// TwinCAT 3 PLC project Untitled1
// ProgramVersion: 3.1.4024.0
// libraries:
//   Tc2_Math, * (Beckhoff Automation GmbH)
//   Tc2_Standard, * (Beckhoff Automation GmbH)
//   Tc2_System, * (Beckhoff Automation GmbH)
//   Tc3_Mc3PlanarMotion, * (Beckhoff Automation GmbH)
//   Tc3_Module, * (Beckhoff Automation GmbH)
//   Tc3_Physics, * (Beckhoff Automation GmbH)
//   XboxControllerUtilities, * (Beckhoff Community)
// project tree:
//   Configuration/ Constraints.TcGVL
//   Mover/ Planar_Mover.TcPOU
//   / PlcTask.TcTTO
//   Controller/ XboxController.TcPOU
// real-time tasks:
//   TASK PlcTask: cycle T#10ms, priority 20, ADS port 350

CONFIGURATION Untitled1
    RESOURCE PLC ON TwinCAT3
        TASK PlcTask(INTERVAL := T#10ms, PRIORITY := 20);
        PROGRAM XboxController WITH PlcTask : XboxController;
        PROGRAM Planar_Mover WITH PlcTask : Planar_Mover;
    END_RESOURCE
END_CONFIGURATION

// ---- Configuration/Constraints.TcGVL
{attribute 'qualified_only'}
VAR_GLOBAL
	

	deltaT						: 		LREAL 	:= 0.000250 ; 	// Cycle time of PLC in Seconds
	maxVelocity					: 		LREAL	:= 150;			// mm/s
	Kp 							:		LREAL      := 3; 		// P Term
	Ki 							:		LREAL      := 0.5; 		// I Term
	Kd 							:		LREAL      := 2; 		// D Term
	Restarting					: 		BOOL;
	
	
END_VAR

// ---- Controller/XboxController.TcPOU
PROGRAM XboxController
VAR

	XboxController1 			: 		FB_Xbox_Controller(NetID := '', iControllerNumber := 1);	
	bIsConnected   				:  		ARRAY [1..2] OF BOOL;
	XpPosition					:		ARRAY [1..2] OF MoverVector; 
	MoverPos					: 		ARRAY [1..2] OF MoverVector;
	invertX						: 		LREAL;
	invertY						: 		LREAL;
	DestinationX				: 		DINT;
	DestinationY				: 		DINT;
	NearestRotationPoint		: 		PositionXYC;
	RotationScailing			: 		LREAL := 0.0002;
	StartTimer					: 		BOOL;
	Timer						: 		TON;
	SnapVAR						: 		BOOL;
	C_VALUE						: 		LREAL;
	MODDED_C					: 		LREAL;
	MoveToC						: 		LREAL;
	ShortestCMove				: 		PositionXYC;
	START						: 		BOOL;
	Ready						: 		BOOL; 
	
	
	
	SanitizedX					: 		LREAL;
	SanitizedY					: 		LREAL;
	SetPointX					: 		REAL;
	SetPointY					: 		REAL;
	ControllerP_Err_X			: 		LREAL;
	ControllerI_Err_X			: 		LREAL;
	ControllerD_Err_X			: 		LREAL;
	ControllerP_Err_Y			: 		LREAL;
	ControllerI_Err_Y			: 		LREAL;
	ControllerD_Err_Y			: 		LREAL;
	PrevSetPointX	 			: 		LREAL;
	PrevSetPointY	 			: 		LREAL;
	PrevSanitizedX				: 		LREAL;
	PrevSanitizedY				: 		LREAL;
	MaxRateOfChange				: 		LREAL;
	IntegralLimit				: 		LREAL;
	MaxIntegralError			: 		LREAL;
	OutputMagnitude				: 		LREAL;
	OutputDirection				: 		LREAL;
	PrevOutputMagnitude			: 		LREAL;
	OutputDistance				: 		LREAL;
	ZeroVector 					: 		MoverVector ;
	nCase						: 		INT := 1;
	Alpha						: 		LREAL := 0.01;
	MaxVelocity					:		LREAL := 10; 
	PastPos10					: 		BOOL;
	PastNeg10					: 		BOOL; 
	BOOL1                       :       BOOL;	
	BOOL2                       :       BOOL;	
	BOOL3						:       BOOL;
	XPoint						: 		BOOL;
	YPoint						: 		BOOL;	
	Height 						: 		LREAL := 2; 
	RESET						:	 	BOOL;
	Go							:		BOOL;
	R_TRIG1						: 		R_TRIG;
	R_TRIG2						: 		R_TRIG;
	SmoothingTon1				:		TON;
	SmoothingTon2				:		TON;
	Ton1						:		TON;
	Ton2						:		TON;
	TRIGGER1					: 		BOOL;
	TRIGGER2					: 		BOOL;
	XPos						: 		INT;
	YPos						: 		INT;
	MaxPosRot					: 		LREAL;
	MaxNegRot					: 		LREAL;
	filtered_output				:	 	LREAL;
	ramp_factor: LREAL;
	ramped_input: LREAL;
	GraphVar: LREAL;
		Prevoutput: LREAL;
		PrevNegRot: LREAL;
	PrevPosRot: LREAL;
		CheckNegRot: LREAL;
	CheckPosRot: LREAL;
		IsUpdated: BOOL;
			Closest90: LREAL;
	
	

END_VAR

//Xbox Controller 1 
XboxController1.Cycle();
bIsConnected[1] := XboxController1.P_Status.bConnected; 

MoverPos[1] := Planar_Mover.fbMover[1].MCTOPLC.ACT.ActPos;

IF Planar_Mover.Done AND NOT ready THEN
	XboxController.init();
END_IF

SetPoint();
		Planar_Mover.fbMover[1].SetExternalSetpoint( XPPosition[1], ZeroVector, ZeroVector);
		
Tilt();
Rotation(); 
ButtonXY();
ButtonA(); 
Bumpers();

METHOD Bumpers 
VAR_INPUT
END_VAR
VAR 
END_VAR

//Hold down for automatic raise and lowering

TON1(IN := XboxController1.P_Buttons.bLeft_Shoulder, PT := T#0.5S); 
TON2(IN := XboxController1.P_Buttons.bRight_Shoulder, PT := T#0.5S); 

IF TON1.Q THEN
	SmoothingTon1.IN := TRUE AND NOT SmoothingTon1.Q;
ELSE
	SmoothingTon1.IN := FALSE;		
END_IF

IF TON2.Q THEN
	SmoothingTon2.IN := TRUE AND NOT SmoothingTon2.Q;
ELSE
	SmoothingTon2.IN := FALSE;
END_IF

//OSR to make sure only one is seen per click 
R_TRIG1(CLK:=XboxController1.P_Buttons.bLeft_Shoulder , Q=> );
R_TRIG2(CLK:=XboxController1.P_Buttons.bRight_Shoulder, Q=> );

IF (R_TRIG1.Q OR SmoothingTon1.Q) AND Height >= -0.35 THEN 
	Height :=  Height - 0.15;
ELSIF (R_TRIG2.Q OR SmoothingTon2.Q) AND Height < 5.0 THEN
	Height := Height + 0.15;
ELSE
	Height := Height; 
END_IF

XpPosition[1].z := Height; 


SmoothingTon1.PT:=T#0.1S;
SmoothingTon2.PT:=T#0.1S;

SmoothingTON1();
SmoothingTON2();
END_METHOD

METHOD buttonA : LREAL
VAR_INPUT
END_VAR
IF XboxController.Ready AND NOT PLanar_Mover.fbMover[1].Error THEN
		
		//Rotation Handeling
		// Find Nearest X
		IF LREAL_TO_INT(MoverPos[1].X) MOD 120 < 60 THEN
			DestinationX	:= 120 * MODTURNS( MoverPos[1].X , 120 );
		ELSE
			DestinationX	:= 120 * (MODTURNS( MoverPos[1].X, 120 ) + 1);
		END_IF
		
		// Find Nearest Y
		IF LREAL_TO_INT(MoverPos[1].Y) MOD 120 < 60 THEN
			DestinationY	:= 120 * MODTURNS( MoverPos[1].Y , 120 );
		ELSE
			DestinationY	:= 120 * (MODTURNS( MoverPos[1].Y, 120 ) + 1);
		END_IF
		
		//Set Boundries for X
		IF DestinationX = 0 THEN
			DestinationX := DestinationX + 120;
		ELSIF DestinationX = 960 THEN
			DestinationX := DestinationX - 120;
		END_IF 	
		
		//Set Boundries for Y
		IF DestinationY = 0 THEN 
			DestinationY := DestinationY + 120;
		ELSIF DestinationY = 720 THEN
			DestinationY := DestinationY - 120;
		END_IF 

		//Move to Nearest Rotation point
			IF XBoxController1.P_Buttons.bA_Button AND MoverPos[1].X < DestinationX THEN
				XpPosition[1].X := XpPosition[1].X + ( 40 * Constraints.deltaT );
			ELSIF XBoxController1.P_Buttons.bA_Button AND MoverPos[1].X > DestinationX THEN
				XpPosition[1].X := XpPosition[1].X -( 40 * Constraints.deltaT );
			END_IF;
			
			IF XBoxController1.P_Buttons.bA_Button AND MoverPos[1].Y < DestinationY THEN
				XpPosition[1].Y := XpPosition[1].Y + ( 40 * Constraints.deltaT );
			ELSIF XBoxController1.P_Buttons.bA_Button AND MoverPos[1].Y > DestinationY THEN
				XpPosition[1].Y := XpPosition[1].Y -( 40 * Constraints.deltaT );
			END_IF;
	
			
			//Checking to make sure Tile is within 1 mm +- of a point that is modulo by 120 and = 0 and then truning a bool true or false
			IF ((LREAL_TO_INT(MoverPos[1].x) MOD 120) >= 119) OR ((LREAL_TO_INT(MoverPos[1].x) MOD 120) <= 1)  THEN
				XPOint := TRUE; 
			ELSE 
				XPoint := FALSE; 
			END_IF
			
			IF ((LREAL_TO_INT(MoverPos[1].y) MOD 120) >= 119) OR ((LREAL_TO_INT(MoverPos[1].y) MOD 120) <= 1) THEN
				YPOint := TRUE; 
			ELSE
				YPoint := FALSE;
			END_IF	
		
		
END_IF
END_METHOD

METHOD buttonXY : LREAL
VAR_INPUT
END_VAR
IF XboxController.Ready AND NOT PLanar_Mover.fbMover[1].Error THEN
	

			//Lock into X movement
		IF XboxController1.P_Buttons.bX_Button THEN
			XpPosition[1].y := XpPosition[1].y ;
		ELSE
			//
		END_IF
		
		//Lock into Y movement
		IF XboxController1.P_Buttons.bY_Button THEN
			XpPosition[1].x := XpPosition[1].x ;
		ELSE
			//
		END_IF
END_IF
END_METHOD

METHOD init 
VAR_INPUT
END_VAR

VAR




END_VAR

IF Planar_mover.MoverState = 3 THEN
	CASE nCase OF 
	1:
		IF Constraints.Restarting THEN
			Constraints.Restarting := FALSE;
			nCase := 4;
		//Wait to Start 
		ELSIF XboxController1.P_Buttons.bStart OR START THEN
			Start := FALSE;
			nCase := 2;
		END_IF
	
	2:
	
	
		//Mover to Play positions
		Planar_Mover.fbMover[1].MoveToPosition(Planar_Mover.cmdFb[1] , Planar_Mover.stMoverPositions[5], Planar_Mover.fbDynMove[1], 0);    
		nCase := 3;
	3:
	
		IF 	Planar_Mover.cmdFB[1].Done THEN
			nCase := 4; 
		END_IF
	
	4:
		//Update Positions
		IF Planar_Mover.cmdFB[1].Done  AND NOT Planar_Mover.cmdFB[1].Busy AND NOT Planar_Mover.cmdFB[2].Busy  THEN
			XpPosition[1].y := MoverPos[1].y; 
			XpPosition[1].x := MoverPos[1].x; 
			XpPosition[1].z := MoverPos[1].z;
			XpPosition[1].c := MoverPos[1].c;
			nCase := 5;
		END_IF
	
	
	5:
	
		//Start External Setpoint Generatior
		Planar_Mover.fbmover[1].StartExternalSetpointGeneration(Planar_Mover.cmdFB[1], Planar_Mover.stExtOptions[1]); 
		nCase := 6; 
	6:
		Ready := TRUE; 
 
		
	END_CASE
ELSIF Planar_Mover.fbMover[1].Error THEN 
	nCase := 1;
	Planar_Mover.fbMover[1].Reset(Planar_Mover.cmdFB[1]); 
	Planar_Mover.init(); 
END_IF
END_METHOD

METHOD rotation : LREAL
VAR_INPUT
END_VAR

VAR






END_VAR
IF XboxController.Ready AND NOT PLanar_Mover.fbMover[1].Error THEN
	
//Holding previous varibles to compare later
PrevNegRot := LREAL_TO_INT(MaxNegRot); 
PrevPosRot := LREAL_TO_INT(MaxPosRot);

//Checking Against previous values 
CheckNegRot := XpPosition[1].c - 10; 
CheckPosRot := XpPosition[1].c + 10; 

// Set the smoothing factor (alpha) and ramping factor (ramp_factor) to values between 0 and 1
alpha := 0.0003;

// Calculate the Filtered value of the input signal
Filtered_Output := alpha * (XboxController1.P_Left_Trigger - XboxController1.P_Right_Trigger) + (1-alpha) * Filtered_Output;

//Actual C
C_VALUE := MoverPos[1].c; 

//Modded C Value
//Make sure to not divide by 0 
IF  C_VALUE <> 0 THEN
	MODDED_C:=MODABS(C_Value,90);
END_IF	
				
		//Endless Rotation 
		IF XPoint AND YPoint THEN
			IF XboxController1.P_Right_Trigger >= 5 AND XboxController1.P_Left_Trigger <= 5 THEN
				//Negative Rotation
				XpPosition[1].c := XpPosition[1].c - (RotationScailing * XboxController1.P_Right_Trigger);
				IsUpdated := FALSE;
			ELSIF XboxController1.P_Left_Trigger >= 5 AND XboxController1.P_Right_Trigger <= 5 THEN
				//Positive Rotation 
				XpPosition[1].c := XpPosition[1].c + (RotationScailing * XboxController1.P_Left_Trigger);
				IsUpdated := FALSE;
			ELSE 
				//Nothing
				IF NOT (PrevNegRot = 0) OR NOT (PrevPosRot = 0) THEN
					IF NOT (isUpdated=TRUE) AND ((PrevNegRot <> CheckNegRot) OR (PrevPosRot <> CheckPosRot)) THEN
						IF Modded_C <= 10 THEN 
							Closest90 := C_Value - Modded_C; 
						ELSIF Modded_C >= 80 THEN
							Closest90 := C_Value + ( 90 - Modded_C);
						END_IF
						MaxNegRot := Closest90 - 10; 
						MaxPosRot := Closest90 + 10;
						IsUpdated := TRUE;
					END_IF
				ELSE
					IF NOT isUpdated THEN
						IF Modded_C <= 10 THEN 
							Closest90 := C_Value - Modded_C; 
						ELSIF Modded_C >= 80 THEN
							Closest90 := C_Value + ( 90 - Modded_C);
						END_IF
						MaxNegRot := Closest90 - 10; 
						MaxPosRot := Closest90 + 10;
						IsUpdated := TRUE; 
					END_IF
				END_IF
			END_IF
		ELSE
			// Apply exponential smoothing to the ramped input signal and limit the output to the range [ActC-10, ActC+10]
			XpPosition[1].c := LIMIT(MaxNegRot, Filtered_Output , MaxPosRot);
		END_IF
		
		
		//Cant move out of rotation point unless within 10 degress 
		IF Modded_C > 10 AND Modded_C < 80 THEN
			PastPos10 := TRUE;
		ELSE 
			PastPos10 := FALSE; 
		END_IF
		

		
		//Set C back to 0
		(*IF XboxController1.P_Left_Trigger >= 98 AND XboxController1.P_Right_Trigger >= 98 THEN
			//Makes sure its intentinal 
			StartTimer := TRUE;
		END_IF*)
		//This simply does not work 
		(*IF Timer.Q THEN 
			IF Modded_C <= 10 THEN 
					Closest90 := C_Value - Modded_C; 
			ELSIF Modded_C >= 80 THEN
					Closest90 := C_Value + ( 90 - Modded_C);
			END_IF
		END_IF *)
		
		
		
END_IF
END_METHOD

METHOD PUBLIC SetPoint 
VAR_INPUT
END_VAR
VAR
	DeltaT: LREAL := 0.000250;
END_VAR
IF XboxController.Ready AND NOT PLanar_Mover.fbMover[1].Error THEN
										
		IF  PastPos10 OR  PastNeg10 THEN
			XPPosition[1].x 	:= XPPosition[1].x  ;
			XPPosition[1].Y 	:= XPPosition[1].Y	;
		ELSE
			invertX				:= SEL(XboxController1.P_Left_Joystick.fX < 1,1,-1);
			invertY				:= SEL(XboxController1.P_Left_Joystick.fY < 1,1,-1);	 
			XPPosition[1].y		:= XPPosition[1].y + (( EXPT(XboxController1.P_Left_Joystick.fY, 2) / 100 )* 4 * deltaT ) * invertY;
			XPPosition[1].x		:= XPPosition[1].x + (( EXPT(XboxController1.P_Left_Joystick.fX, 2) / 100 )* 4 * deltaT ) * invertX;
		END_IF
		

ELSIF Planar_Mover.fbMover[1].Error THEN
	Ready := FALSE; 
	Planar_Mover.fbMover[1].Reset(Planar_Mover.cmdFB[1]);  
	PLanar_mover.init(); 
END_IF
END_METHOD

METHOD Tilt : LREAL
VAR_INPUT
END_VAR
IF XboxController.Ready AND NOT PLanar_Mover.fbMover[1].Error THEN
			//A tilt 
		XPPosition[1].a		:= 0.008 * XboxController1.p_Right_Joystick.fY;
		
		//B tilt 	
		XPPosition[1].b   	:= 0.008 * XboxController1.p_Right_Joystick.fX; 
END_IF
END_METHOD

END_PROGRAM

// ---- Mover/Planar_Mover.TcPOU
PROGRAM Planar_Mover
VAR
	
fbMover 					:		ARRAY [1..2]  OF MC_PlanarMover ; // Change based on how many movers there are
cmdFB 						:		ARRAY [1..2]  OF MC_PlanarFeedBack ; 
stMoverPositions 			:		ARRAY [1..12] OF PositionXYC ;
fbDynMove					:		ARRAY [1..5]  OF DynamicConstraint_PathXY ;
stExtOptions				:		ARRAY [1..2]  OF ST_ExternalSetpointGenerationOptions; 
Done						: 	 	BOOL;
nCase						: 		INT := 1;
timer						: 		TON;
moverState					:		MC_Planar_State; 
RESET						: 		BOOL;


END_VAR

//Mover 1 updates
fbMover[1].Update(); 
cmdFB[1].Update();
moverState := fbMover[1].MCTOPLC.STD.State;

Timer(IN := TRUE, PT := T#1S); 

IF Timer.Q THEN
	//Start initizalization
	IF NOT done OR MoverState = 5 OR MoverState = 1 THEN 
		Planar_Mover.init();
	END_IF 
END_IF

METHOD init 
VAR_INPUT
END_VAR

VAR


END_VAR
CASE nCase OF
1: 
	//fbmover[1].StopExternalSetpointGeneration(cmdFb[1]);
	Done := FALSE;
	fbMover[1].Reset(cmdFB[1]);
	//fbMover[2].Reset(cmdFB[2]);
	nCase := 2;

2:

	IF cmdFB[1].Done THEN
		nCase := 3; 
	END_IF
	
3:

	fbMover[1].Enable(cmdFB[1]);
	nCase := 4;
	
4:

	IF cmdFB[1].Done THEN
		nCase := 5;
	END_IF
	
5:

//Set up Case
	// Setting Movingg Positions 
	stMoverPositions[5].SetValuesXYC(120,360,0); // Mover 1 Start 

	// Normal Movememnt
	fbDynMove[1].SetValuesVADJ(500,5000,5000,20000); // Normal
	fbDynMove[2].SetValuesVADJ(1000,5000,5000,20000);// Fast
	fbDynMove[3].SetValuesVADJ(200,2000,5000,10000); // Slow

	stExtOptions[1].mode := MC_EXTERNAL_SET_POSITION_MODE.Absolute; // Setting up external Setpoint generator
	nCase := 6; 
6:

Done := TRUE; 
nCase := 7;

7:

IF MoverState = 5 OR MoverState = 1 THEN
	IF XboxController.XboxController1.P_Buttons.bBack OR RESET THEN
		Constraints.Restarting := TRUE;  
		nCase := 1;	
	END_IF
END_IF 

	
END_CASE
END_METHOD

END_PROGRAM
